Staubli VAL3: RobotStateMsg.dtx

public bool bIsInitialized = true
public MessageHeader header
public RobotState robotState
public num nSerializedData
